FUNCTION_BLOCK DP (* Diagnostic Point *)
  (* Standard: 61499-2; ApplicationDomain: Fault Diagnostics; Function: Interface to the agents in the Multiagent Fault Diagnostic Engine (FDE).; Type: Composite Function Block; Description: The DP function block operates as a probe that allows a FDE agent to interact with a function block from the inside of the function block application. *)
  (* Version 1.0, 2020-05-28, Badger, AUT *)
  (* Compiler Cpp Unknown Unknown 1.0 *)
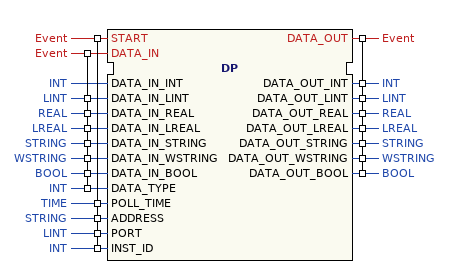
  EVENT_INPUT
    START WITH ADDRESS, PORT, INST_ID, POLL_TIME;
    DATA_IN WITH DATA_IN_BOOL, DATA_TYPE, DATA_IN_WSTRING, DATA_IN_STRING, DATA_IN_LREAL, DATA_IN_REAL, DATA_IN_LINT; (* Normal Execution Request *)
  END_EVENT
  EVENT_OUTPUT
    DATA_OUT WITH DATA_OUT_BOOL, DATA_OUT_INT, DATA_OUT_LINT, DATA_OUT_REAL, DATA_OUT_LREAL, DATA_OUT_STRING, DATA_OUT_WSTRING; (* Initialization Confirm *)
  END_EVENT
  VAR_INPUT
    DATA_IN_INT : INT;
    DATA_IN_LINT : LINT;
    DATA_IN_REAL : REAL;
    DATA_IN_LREAL : LREAL;
    DATA_IN_STRING : STRING;
    DATA_IN_WSTRING : WSTRING;
    DATA_IN_BOOL : BOOL; (* Input event qualifier *)
    DATA_TYPE : INT;
    POLL_TIME : TIME;
    ADDRESS : STRING;
    PORT : LINT;
    INST_ID : INT;
  END_VAR
  VAR_OUTPUT
    DATA_OUT_INT : INT;
    DATA_OUT_LINT : LINT;
    DATA_OUT_REAL : REAL;
    DATA_OUT_LREAL : LREAL;
    DATA_OUT_STRING : STRING;
    DATA_OUT_WSTRING : WSTRING;
    DATA_OUT_BOOL : BOOL; (* Output event qualifier *)
  END_VAR
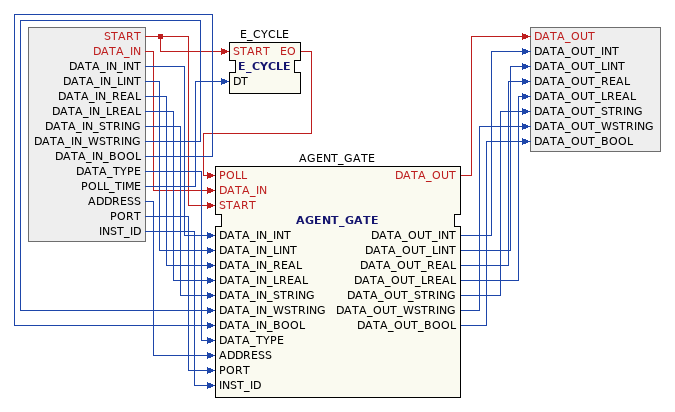
  FBS
    E_CYCLE : E_CYCLE;
    AGENT_GATE : AGENT_GATE;
  END_FBS
  EVENT_CONNECTIONS
    START TO E_CYCLE.START;
    E_CYCLE.EO TO AGENT_GATE.POLL;
    DATA_IN TO AGENT_GATE.DATA_IN;
    AGENT_GATE.DATA_OUT TO DATA_OUT;
    START TO AGENT_GATE.START;
  END_CONNECTIONS
  DATA_CONNECTIONS
    POLL_TIME TO E_CYCLE.DT;
    DATA_IN_INT TO AGENT_GATE.DATA_IN_INT;
    DATA_IN_LINT TO AGENT_GATE.DATA_IN_LINT;
    DATA_IN_REAL TO AGENT_GATE.DATA_IN_REAL;
    DATA_IN_LREAL TO AGENT_GATE.DATA_IN_LREAL;
    DATA_IN_STRING TO AGENT_GATE.DATA_IN_STRING;
    DATA_IN_WSTRING TO AGENT_GATE.DATA_IN_WSTRING;
    DATA_IN_BOOL TO AGENT_GATE.DATA_IN_BOOL;
    DATA_TYPE TO AGENT_GATE.DATA_TYPE;
    ADDRESS TO AGENT_GATE.ADDRESS;
    PORT TO AGENT_GATE.PORT;
    INST_ID TO AGENT_GATE.INST_ID;
    AGENT_GATE.DATA_OUT_INT TO DATA_OUT_INT;
    AGENT_GATE.DATA_OUT_LINT TO DATA_OUT_LINT;
    AGENT_GATE.DATA_OUT_REAL TO DATA_OUT_REAL;
    AGENT_GATE.DATA_OUT_LREAL TO DATA_OUT_LREAL;
    AGENT_GATE.DATA_OUT_STRING TO DATA_OUT_STRING;
    AGENT_GATE.DATA_OUT_WSTRING TO DATA_OUT_WSTRING;
    AGENT_GATE.DATA_OUT_BOOL TO DATA_OUT_BOOL;
  END_CONNECTIONS
END_FUNCTION_BLOCK
